// Mitsubishi GX Works2 project: Group_32_14.5_run1   PLC: FX3G

// global labels: Global1
VAR_GLOBAL
  StartDay AT X007 : BOOL;
  RaspberryInput AT D1110 : INT;
  RaspberryInventory AT D1100 : INT;
  LemonInput AT D1112 : INT;
  LemonInventory AT D1102 : INT;
  GummyInput AT D1118 : INT;
  GummyInventory AT D1106 : INT;
  StabilizerInput AT D1114 : INT;
  StabilizerInventory AT D1104 : INT;
  StartPrep AT X001 : BOOL;
  StartCooling AT X002 : BOOL;
  CoolSensor AT X003 : BOOL;
  AnalogOutput AT D8282 : INT;
  SwitchesOff AT M40 : BOOL;
  Outputstorage AT D1160 : INT;
  WorkDay AT Y007 : BOOL;
  AnalogInput1 AT D8280 : INT;
END_VAR
VAR_GLOBAL CONSTANT
  Constant5 : INT := 5;
END_VAR
VAR_GLOBAL
  TypeRegular AT M2 : BOOL;
  TypeLuxury AT M3 : BOOL;
END_VAR
VAR_GLOBAL CONSTANT
  RaspberryMinReqR : INT := 280;
  LemonMinReqR : INT := 455;
  GummyMinReqR : INT := 25;
  StabilizerMinReqR : INT := 105;
  LemonMinReqL : INT := 665;
  RaspberryMinReqL : INT := 385;
  GummyMinReqL : INT := 70;
  StabilizerMinReqL : INT := 210;
END_VAR
VAR_GLOBAL
  GotRaspberry AT M4 : BOOL;
  GotLemon AT M5 : BOOL;
  GotStabilizer AT M6 : BOOL;
  GotGummy AT M7 : BOOL;
  EnoughStock AT M1 : BOOL;
  EndWorkDay AT M10 : BOOL;
  Emergency AT X005 : BOOL;
  NewIteration AT M8 : BOOL;
  IterationGoing AT M9 : BOOL;
  PrepLight AT Y000 : BOOL;
END_VAR
VAR_GLOBAL CONSTANT
  Const5Sec : INT := 50;
  RaspberryContR : INT := 350;
  LemonContR : INT := 490;
  RaspberryContL : INT := 560;
  LemonContL : INT := 700;
END_VAR
VAR_GLOBAL
  RaspberryCreamCont AT D1120 : INT;
  LemonCreamCont AT D1122 : INT;
  FinishCream AT M50 : BOOL;
  PerpTimerFinished AT TS1 : BOOL;
  CastingTimer AT TC1 : BOOL;
  PrepTimer AT TC1 : BOOL;
  FinishPrepProcess AT M51 : BOOL;
  RaspberryCoolCont AT D1124 : INT;
  LemonCoolCont AT D1126 : INT;
  FinishMoveToCool AT M52 : BOOL;
  CoolLight AT Y002 : BOOL;
  CoolTimer AT TC2 : BOOL;
END_VAR
VAR_GLOBAL CONSTANT
  Const8Sec : INT := 80;
END_VAR
VAR_GLOBAL
  FinishCool AT TS2 : BOOL;
  MixCont AT D1130 : INT;
  FinishMoveToMix AT M53 : BOOL;
END_VAR
VAR_GLOBAL CONSTANT
  GummyContR : INT := 4;
  GummyContL : INT := 10;
END_VAR
VAR_GLOBAL
  MixTimer_R AT TC3 : BOOL;
  MixTimerDone_R AT TS3 : BOOL;
  MixTimer_L AT TC4 : BOOL;
  MixTimerDone_L AT TS4 : BOOL;
  MixLight1 AT Y005 : BOOL;
  MixLight2 AT Y006 : BOOL;
  FinishMix AT M54 : BOOL;
END_VAR
VAR_GLOBAL CONSTANT
  Const3SecMix : INT := 30;
  Const5secMix : INT := 50;
END_VAR
VAR_GLOBAL
  MixFlashing AT M55 : BOOL;
  Bulb5Timer AT TC5 : BOOL;
  Bulb5Finish AT TS5 : BOOL;
  Bulb6Timer AT TC6 : BOOL;
  Bulb6Finish AT TS6 : BOOL;
END_VAR
VAR_GLOBAL CONSTANT
  FlashConst : INT := 10;
END_VAR
VAR_GLOBAL
  bulb5 AT Y005 : BOOL;
  bulb6 AT Y006 : BOOL;
  IcecreamInPackageCounter AT CC7 : BOOL;
  PackingIdicator AT M20 : BOOL;
  StartPacking AT X000 : BOOL;
  IcecreamPacked AT CS7 : BOOL;
  IcecreamPack7 AT K7 : INT;
END_VAR
VAR_GLOBAL CONSTANT
  Cons40 : INT := 40;
END_VAR
VAR_GLOBAL
  Test AT M70 : BOOL;
  TestLight AT Y011 : BOOL;
  CoolSensorLight AT M45 : BOOL;
  CoolSensorLight2 AT M46 : BOOL;
  FinishIteration AT M21 : BOOL;
END_VAR

// task Task_01 (event TRUE, interval 0, priority 31): POU_01

PROGRAM POU_01
(* structured ladder/FBD written out as ST: instructions are called as NAME(EN, inputs, outputs); _pN, _eN, _tN stand for wires *)
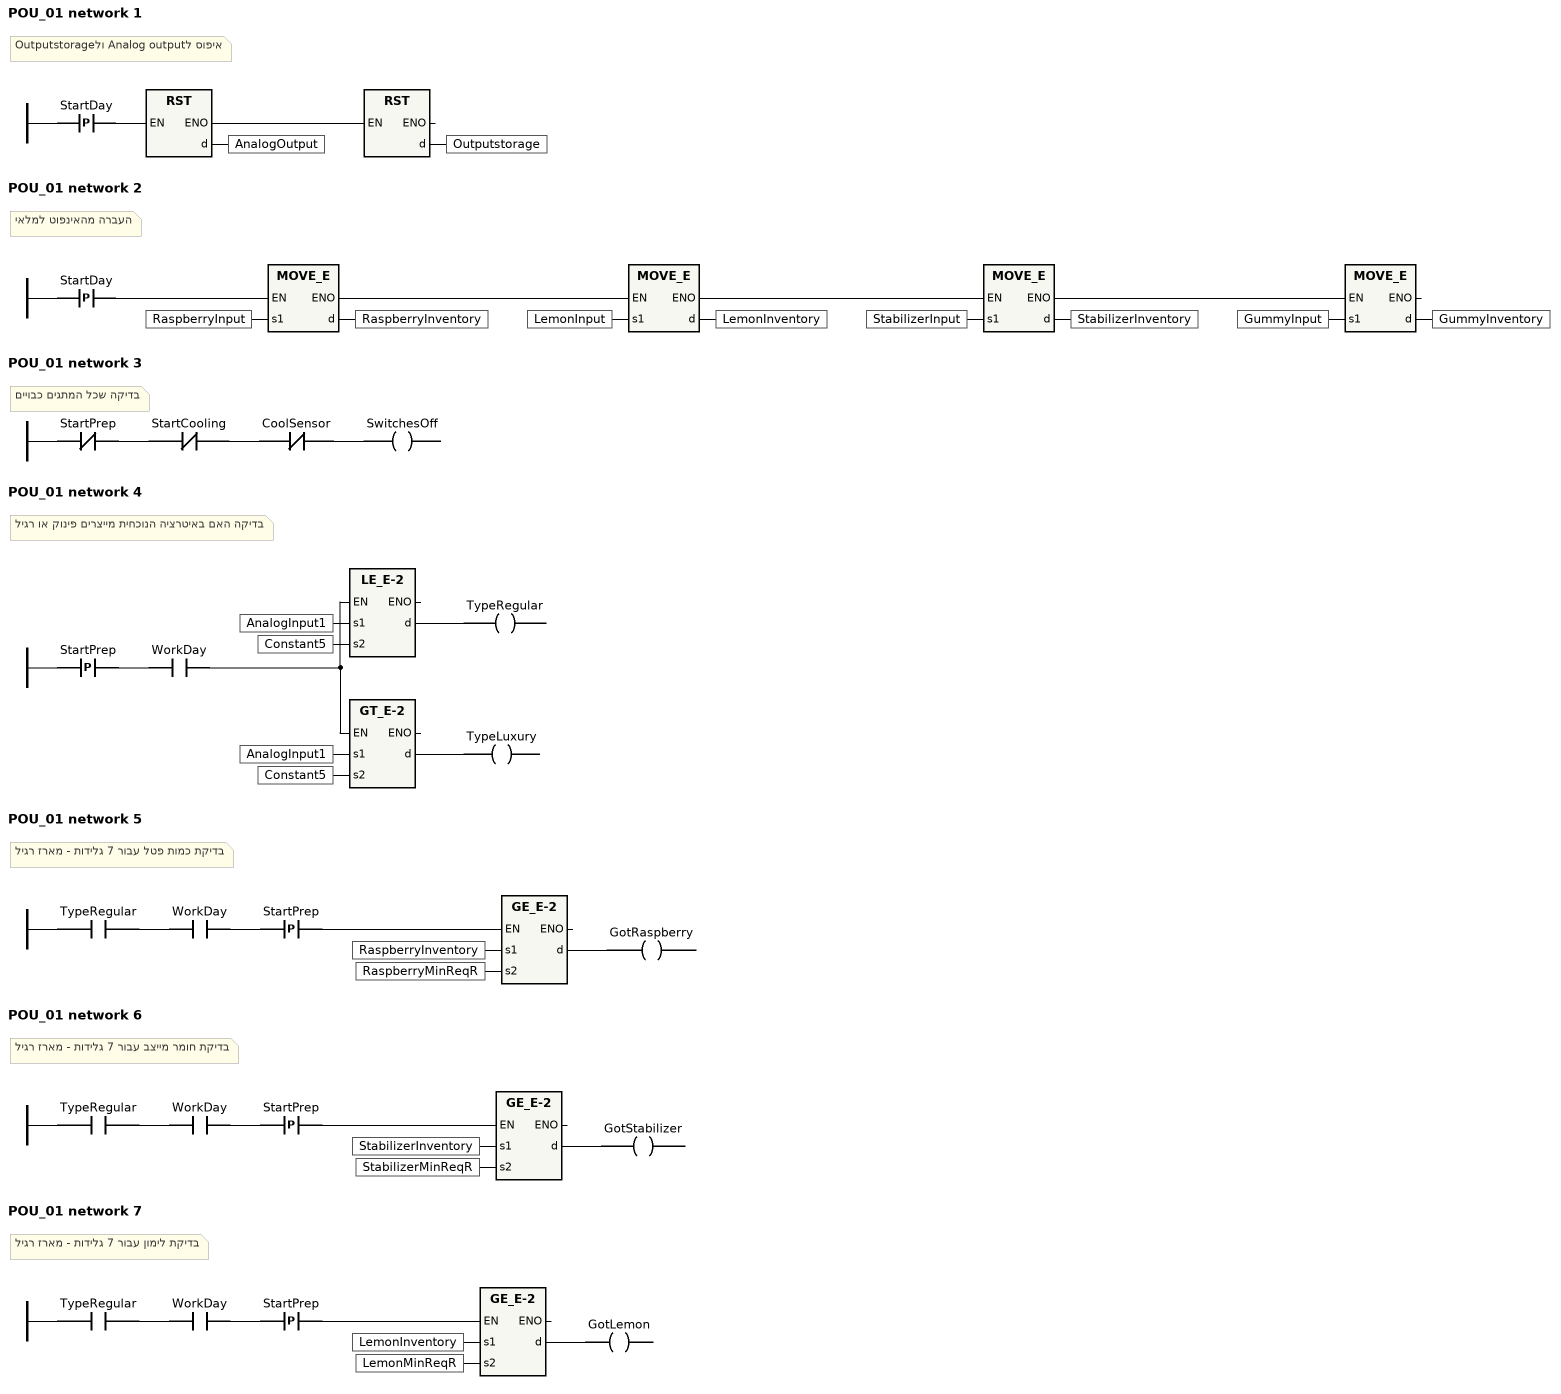
(* network 1 *)
(* איפוס לAnalog output ולOutputstorage *)
_e1 := RST(LDP(TRUE, StartDay), AnalogOutput);
RST(_e1, Outputstorage);
(* network 2 *)
(* העברה מהאינפוט למלאי *)
_e1 := MOVE_E(LDP(TRUE, StartDay), RaspberryInput, RaspberryInventory);
_e2 := MOVE_E(_e1, LemonInput, LemonInventory);
_e3 := MOVE_E(_e2, StabilizerInput, StabilizerInventory);
MOVE_E(_e3, GummyInput, GummyInventory);
(* network 3 *)
(* בדיקה שכל המתגים כבויים *)
SwitchesOff := NOT StartPrep AND NOT StartCooling AND NOT CoolSensor;
(* network 4 *)
(* בדיקה האם באיטרציה הנוכחית מייצרים פינוק או רגיל *)
_p1 := LDP(TRUE, StartPrep) AND WorkDay;
LE_E(_p1, AnalogInput1, Constant5, _t2);
TypeRegular := _t2;
GT_E(_p1, AnalogInput1, Constant5, _t3);
TypeLuxury := _t3;
(* network 5 *)
(* בדיקת כמות פטל עבור 7 גלידות - מארז רגיל *)
GE_E(TypeRegular AND WorkDay AND LDP(TRUE, StartPrep), RaspberryInventory, RaspberryMinReqR, _t1);
GotRaspberry := _t1;
(* network 6 *)
(* בדיקת חומר מייצב עבור 7 גלידות - מארז רגיל *)
GE_E(TypeRegular AND WorkDay AND LDP(TRUE, StartPrep), StabilizerInventory, StabilizerMinReqR, _t1);
GotStabilizer := _t1;
(* network 7 *)
(* בדיקת לימון עבור 7 גלידות - מארז רגיל *)
GE_E(TypeRegular AND WorkDay AND LDP(TRUE, StartPrep), LemonInventory, LemonMinReqR, _t1);
GotLemon := _t1;
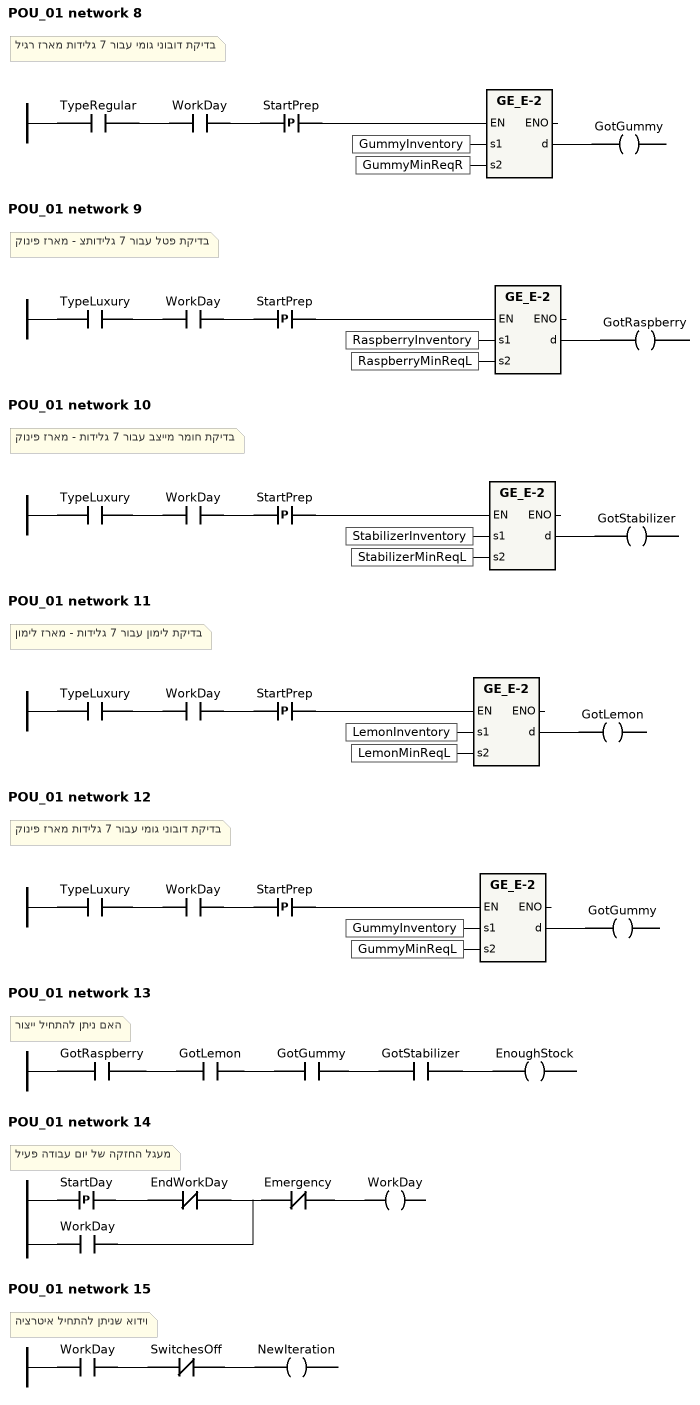
(* network 8 *)
(* בדיקת דובוני גומי עבור 7 גלידות מארז רגיל *)
GE_E(TypeRegular AND WorkDay AND LDP(TRUE, StartPrep), GummyInventory, GummyMinReqR, _t1);
GotGummy := _t1;
(* network 9 *)
(* בדיקת פטל עבור 7 גלידותצ - מארז פינוק *)
GE_E(TypeLuxury AND WorkDay AND LDP(TRUE, StartPrep), RaspberryInventory, RaspberryMinReqL, _t1);
GotRaspberry := _t1;
(* network 10 *)
(* בדיקת חומר מייצב עבור 7 גלידות - מארז פינוק *)
GE_E(TypeLuxury AND WorkDay AND LDP(TRUE, StartPrep), StabilizerInventory, StabilizerMinReqL, _t1);
GotStabilizer := _t1;
(* network 11 *)
(* בדיקת לימון עבור 7 גלידות - מארז לימון *)
GE_E(TypeLuxury AND WorkDay AND LDP(TRUE, StartPrep), LemonInventory, LemonMinReqL, _t1);
GotLemon := _t1;
(* network 12 *)
(* בדיקת דובוני גומי עבור 7 גלידות מארז פינוק *)
GE_E(TypeLuxury AND WorkDay AND LDP(TRUE, StartPrep), GummyInventory, GummyMinReqL, _t1);
GotGummy := _t1;
(* network 13 *)
(* האם ניתן להתחיל ייצור *)
EnoughStock := GotRaspberry AND GotLemon AND GotGummy AND GotStabilizer;
(* network 14 *)
(* מעגל החזקה של יום עבודה פעיל *)
WorkDay := ((LDP(TRUE, StartDay) AND NOT EndWorkDay) OR WorkDay) AND NOT Emergency;
(* network 15 *)
(* וידוא שניתן להתחיל איטרציה *)
NewIteration := WorkDay AND NOT SwitchesOff;
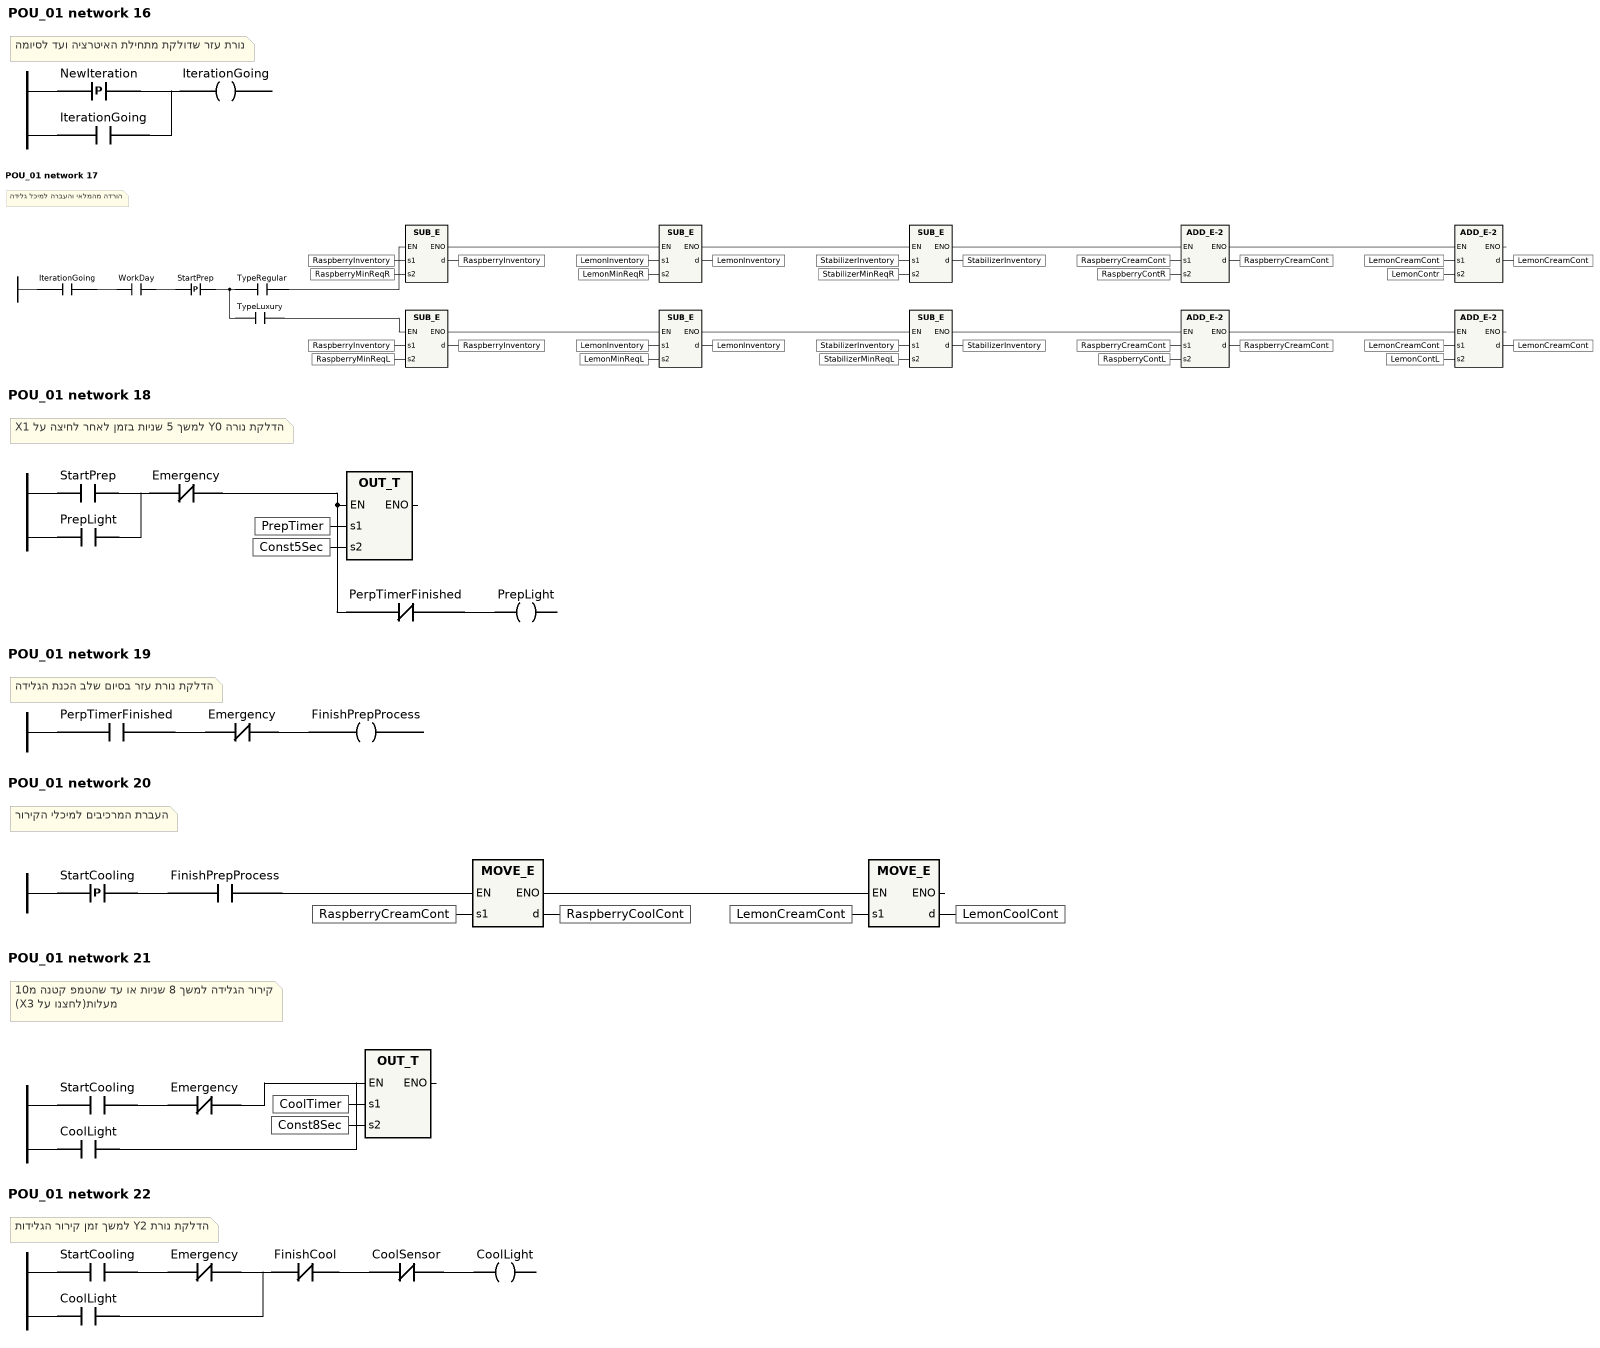
(* network 16 *)
(* נורת עזר שדולקת מתחילת האיטרציה ועד לסיומה *)
IterationGoing := LDP(TRUE, NewIteration) OR IterationGoing;
(* network 17 *)
(* הורדה מהמלאי והעברה למיכל גלידה *)
_p1 := IterationGoing AND WorkDay AND LDP(TRUE, StartPrep);
_e2 := SUB_E(_p1 AND TypeRegular, RaspberryInventory, RaspberryMinReqR, RaspberryInventory);
_e3 := SUB_E(_e2, LemonInventory, LemonMinReqR, LemonInventory);
_e4 := SUB_E(_e3, StabilizerInventory, StabilizerMinReqR, StabilizerInventory);
_e5 := ADD_E(_e4, RaspberryCreamCont, RaspberryContR, RaspberryCreamCont);
ADD_E(_e5, LemonCreamCont, LemonContr, LemonCreamCont);
_e6 := SUB_E(_p1 AND TypeLuxury, RaspberryInventory, RaspberryMinReqL, RaspberryInventory);
_e7 := SUB_E(_e6, LemonInventory, LemonMinReqL, LemonInventory);
_e8 := SUB_E(_e7, StabilizerInventory, StabilizerMinReqL, StabilizerInventory);
_e9 := ADD_E(_e8, RaspberryCreamCont, RaspberryContL, RaspberryCreamCont);
ADD_E(_e9, LemonCreamCont, LemonContL, LemonCreamCont);
(* network 18 *)
(* הדלקת נורה Y0 למשך 5 שניות בזמן לאחר לחיצה על X1 *)
_p1 := (StartPrep OR PrepLight) AND NOT Emergency;
PrepLight := _p1 AND NOT PerpTimerFinished;
OUT_T(_p1, PrepTimer, Const5Sec);
(* network 19 *)
(* הדלקת נורת עזר בסיום שלב הכנת הגלידה *)
FinishPrepProcess := PerpTimerFinished AND NOT Emergency;
(* network 20 *)
(* העברת המרכיבים למיכלי הקירור *)
_e1 := MOVE_E(LDP(TRUE, StartCooling) AND FinishPrepProcess, RaspberryCreamCont, RaspberryCoolCont);
MOVE_E(_e1, LemonCreamCont, LemonCoolCont);
(* network 21 *)
(* קירור הגלידה למשך 8 שניות או עד שהטמפ קטנה מ10 מעלות(לחצנו על X3) *)
OUT_T((StartCooling AND NOT Emergency) OR CoolLight, CoolTimer, Const8Sec);
(* network 22 *)
(* הדלקת נורת Y2 למשך זמן קירור הגלידות *)
CoolLight := (((StartCooling AND NOT Emergency) OR CoolLight) AND NOT FinishCool) AND NOT CoolSensor;
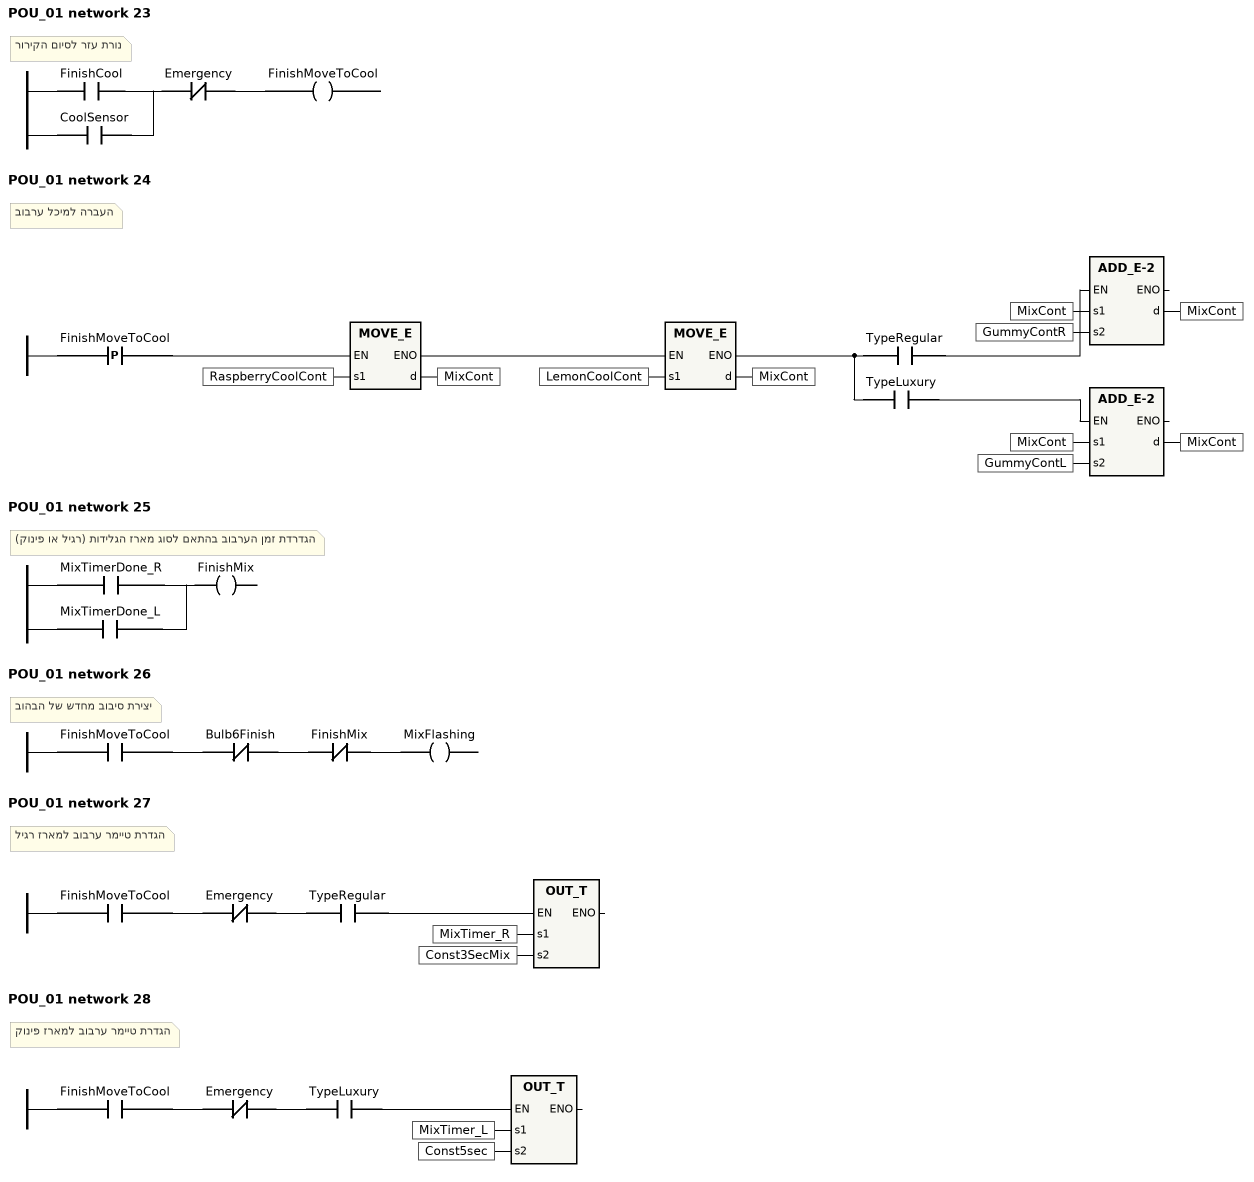
(* network 23 *)
(* נורת עזר לסיום הקירור *)
FinishMoveToCool := (FinishCool OR CoolSensor) AND NOT Emergency;
(* network 24 *)
(* העברה למיכל ערבוב *)
_e1 := MOVE_E(LDP(TRUE, FinishMoveToCool), RaspberryCoolCont, MixCont);
_e2 := MOVE_E(_e1, LemonCoolCont, MixCont);
ADD_E(_e2 AND TypeRegular, MixCont, GummyContR, MixCont);
ADD_E(_e2 AND TypeLuxury, MixCont, GummyContL, MixCont);
(* network 25 *)
(* הגדרדת זמן הערבוב בהתאם לסוג מארז הגלידות (רגיל או פינוק) *)
FinishMix := MixTimerDone_R OR MixTimerDone_L;
(* network 26 *)
(* יצירת סיבוב מחדש של הבהוב *)
MixFlashing := FinishMoveToCool AND NOT Bulb6Finish AND NOT FinishMix;
(* network 27 *)
(* הגדרת טיימר ערבוב למארז רגיל *)
OUT_T(FinishMoveToCool AND NOT Emergency AND TypeRegular, MixTimer_R, Const3SecMix);
(* network 28 *)
(* הגדרת טיימר ערבוב למארז פינוק *)
OUT_T(FinishMoveToCool AND NOT Emergency AND TypeLuxury, MixTimer_L, Const5sec);
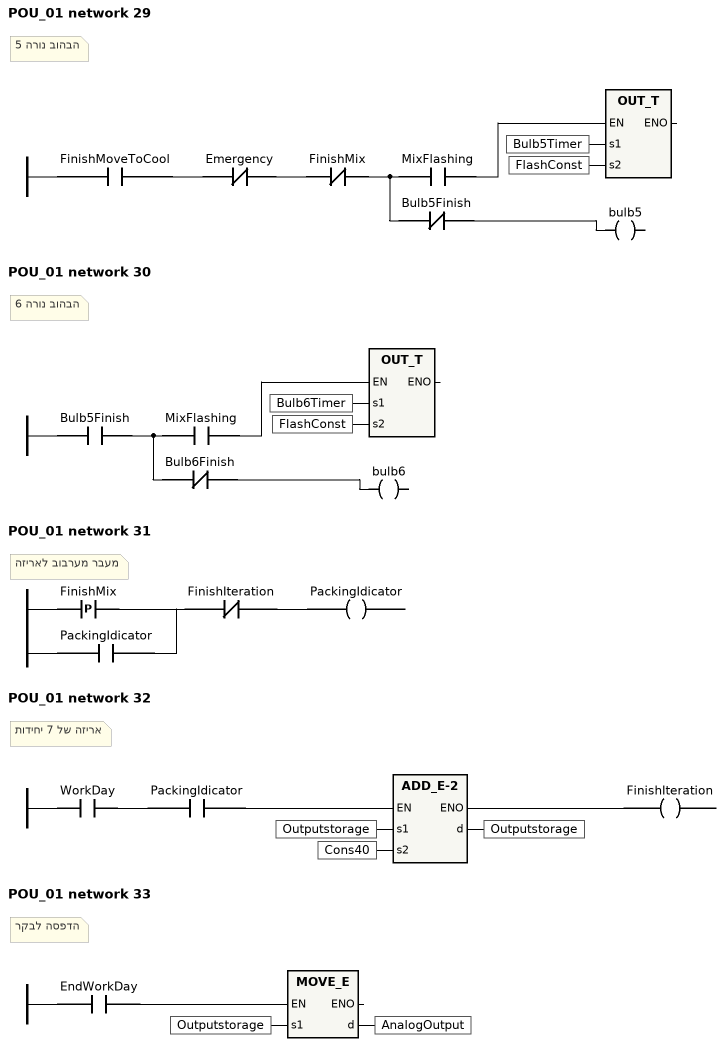
(* network 29 *)
(* הבהוב נורה 5 *)
_p1 := FinishMoveToCool AND NOT Emergency AND NOT FinishMix;
OUT_T(_p1 AND MixFlashing, Bulb5Timer, FlashConst);
bulb5 := _p1 AND NOT Bulb5Finish;
(* network 30 *)
(* הבהוב נורה 6 *)
OUT_T(Bulb5Finish AND MixFlashing, Bulb6Timer, FlashConst);
bulb6 := Bulb5Finish AND NOT Bulb6Finish;
(* network 31 *)
(* מעבר מערבוב לאריזה *)
PackingIdicator := (LDP(TRUE, FinishMix) OR PackingIdicator) AND NOT FinishIteration;
(* network 32 *)
(* אריזה של 7 יחידות *)
_e1 := ADD_E(WorkDay AND PackingIdicator, Outputstorage, Cons40, Outputstorage);
FinishIteration := _e1;
(* network 33 *)
(* הדפסה לבקר *)
MOVE_E(EndWorkDay, Outputstorage, AnalogOutput);
END_PROGRAM
